// TIA Portal V16 program export: 1 tag tables, 12 data types, 26 data blocks, 18 code blocks (in call order from the OBs), 1 instance data blocks

VAR_GLOBAL   // PLC tag table "Default tag table"
   io_a AT %I0.0 : Bool;
   io_b AT %I0.1 : Bool;
END_VAR
VAR_GLOBAL CONSTANT   // user constants
   MAX_RPM : Int := 2800;
END_VAR

TYPE "SensorCommand"
VERSION : 0.1
   STRUCT
      enable { ExternalAccessible := 'False'; ExternalVisible := 'False'; ExternalWritable := 'False'} : Bool;
      mute { ExternalAccessible := 'False'; ExternalVisible := 'False'; ExternalWritable := 'False'} : Bool;
      case { ExternalAccessible := 'False'; ExternalVisible := 'False'; ExternalWritable := 'False'} : Int;
   END_STRUCT;

END_TYPE

TYPE "AnonStruct"
VERSION : 0.1
   STRUCT
      command : Struct
         a : Bool;
         b : Bool;
         c : Bool;
         others : Struct
            x : Bool;
            y : Bool;
            z : Bool := true;   // Definitely keep this one on.
         END_STRUCT;
      END_STRUCT;
   END_STRUCT;

END_TYPE

TYPE "ArrayWithDefault"
VERSION : 0.1
   STRUCT
      v : Array[0..15] of Bool := [false, true];
   END_STRUCT;

END_TYPE

TYPE "Pointf"
VERSION : 0.1
   STRUCT
      x : Real;
      y : Real;
   END_STRUCT;

END_TYPE

TYPE "Pointi"
VERSION : 0.1
   STRUCT
      x : Int;
      y : Int;
   END_STRUCT;

END_TYPE

TYPE "Polygon"
VERSION : 0.1
   STRUCT
      vertices { S7_SetPoint := 'False'} : Array[0..9] of "Pointi";   // Fixed size array
      n { S7_SetPoint := 'True'} : Int;   // of which this many points are valid
   END_STRUCT;

END_TYPE

TYPE "AppControl"
VERSION : 0.1
   STRUCT
      start : Bool;
      stop : Bool;
   END_STRUCT;

END_TYPE

TYPE "Box"
VERSION : 0.1
   STRUCT
      min { S7_SetPoint := 'False'} : "Point";
      max { S7_SetPoint := 'False'} : "Point";
   END_STRUCT;

END_TYPE

TYPE "MachineState"
VERSION : 0.1
   STRUCT
      running : Bool;
      faulted : Bool;
   END_STRUCT;

END_TYPE

TYPE "Point"
VERSION : 0.1
   STRUCT
      x : Int;
      y : Int;
   END_STRUCT;

END_TYPE

TYPE "SensorControl"
VERSION : 0.1
   STRUCT
      request_mode : Int;
   END_STRUCT;

END_TYPE

TYPE "SensorState"
VERSION : 0.1
   STRUCT
      mode : Int;
      ready : Bool;
   END_STRUCT;

END_TYPE

DATA_BLOCK "FromSafety"   // DB3
{ S7_Optimized_Access := 'TRUE' }
VERSION : 0.1
// stored: AutoNumber true, DBAccessibleFromOPCUA true, IsOnlyStoredInLoadMemory false, IsRetainMemResEnabled false, IsWriteProtectedInAS false, MemoryReserve 100
   VAR
      stop : Bool;
   END_VAR
BEGIN
END_DATA_BLOCK

DATA_BLOCK "ToSafety"   // DB2
{ S7_Optimized_Access := 'TRUE' }
VERSION : 0.1
// stored: AutoNumber true, DBAccessibleFromOPCUA true, IsOnlyStoredInLoadMemory false, IsRetainMemResEnabled false, IsWriteProtectedInAS false, MemoryReserve 100
   VAR
      "a" : Bool;
      "b" : Bool;
   END_VAR
BEGIN
END_DATA_BLOCK

DATA_BLOCK "DebugData"
{ S7_Optimized_Access := "TRUE" }
VERSION: 0.1
NON_RETAIN
    VAR
        source { ExternalAccessible := 'False'; ExternalVisible := 'False'; ExternalWritable := 'False'} : Int;
        flag : Bool;
    END_VAR

BEGIN
    source := 1;

END_DATA_BLOCK

DATA_BLOCK "AnonTestDB"
{ S7_Optimized_Access := 'TRUE' }
VERSION : 0.1
NON_RETAIN
   VAR 
      a { S7_SetPoint := 'False'} : "AnonStruct";
      b : "AnonStruct";   // custom comment for b
   END_VAR


BEGIN

END_DATA_BLOCK

DATA_BLOCK "PolygonDB"
{ S7_Optimized_Access := 'TRUE' }
VERSION : 0.1
NON_RETAIN
"Polygon"

BEGIN
   vertices[0].x := 0;
   vertices[0].y := 0;

END_DATA_BLOCK

DATA_BLOCK "DataFromSafety"
{ S7_Optimized_Access := 'TRUE' }
VERSION : 0.1
NON_RETAIN
   VAR 
      running : Bool;
   END_VAR


BEGIN

END_DATA_BLOCK

DATA_BLOCK "DataToSafety"
{ S7_Optimized_Access := 'TRUE' }
VERSION : 0.1
NON_RETAIN
   VAR 
      run : Bool;
   END_VAR


BEGIN

END_DATA_BLOCK

DATA_BLOCK "Main_Safety_RTG1_DB"
{ S7_Optimized_Access := 'TRUE' }
NAME : FUSI
VERSION : 0.1
NON_RETAIN
"Main_Safety_RTG1"

BEGIN

END_DATA_BLOCK

DATA_BLOCK "BlockIncrementer_DB"
{ S7_Optimized_Access := 'TRUE' }
VERSION : 0.1
NON_RETAIN
"BlockIncrementer"

BEGIN

END_DATA_BLOCK

DATA_BLOCK "MyCounter_DB0"
{ S7_Optimized_Access := 'TRUE' }
VERSION : 0.1
NON_RETAIN
"MyCounter"

BEGIN

END_DATA_BLOCK

DATA_BLOCK "MyCounter_DB1"
{ S7_Optimized_Access := 'TRUE' }
VERSION : 0.1
NON_RETAIN
"MyCounter"

BEGIN

END_DATA_BLOCK

DATA_BLOCK "Box"
{ S7_Optimized_Access := 'TRUE' }
VERSION : 0.1
NON_RETAIN
"Box"

BEGIN
   min.x := 0;

END_DATA_BLOCK

DATA_BLOCK "Example1_DB"
{ S7_Optimized_Access := 'TRUE' }
VERSION : 0.1
NON_RETAIN
   VAR 
      box0 { S7_SetPoint := 'False'} : "Box";
      box1 : "Box";
   END_VAR


BEGIN

END_DATA_BLOCK

DATA_BLOCK "Example2_DB"
{ S7_Optimized_Access := 'TRUE' }
VERSION : 0.1
NON_RETAIN
   VAR 
      reference { ExternalAccessible := 'False'; ExternalVisible := 'False'; ExternalWritable := 'False'; S7_SetPoint := 'False'} : "Point";
   END_VAR


BEGIN
   reference.x := 0;
   reference.y := 1;

END_DATA_BLOCK

DATA_BLOCK "F_SystemInfo_DB"
{ S7_Optimized_Access := 'TRUE' }
NAME : F_GLOBDB
VERSION : 0.1
NON_RETAIN
   VAR 
      FCCValue : DWord;
   END_VAR


BEGIN

END_DATA_BLOCK

DATA_BLOCK "RTG1SysInfo"
{InstructionName := 'F_CTRL1';
 LibVersion := '2.2';
 S7_Optimized_Access := 'TRUE' }
AUTHOR : SafeSys
FAMILY : F_CTRL
NAME : F_CTRL_1
VERSION : 2.2
NON_RETAIN
F_CTRL1

BEGIN
   F_SYSINFO.F_PROG_SIG := DW#16#832DEE38;
   F_SYSINFO.F_PROG_DAT := DTL#2021-8-4-22:50:56.862582800;
   F_SYSINFO.F_RTG_SIG := DW#16#F5BD20EF;
   F_SYSINFO.F_RTG_DAT := DTL#2021-8-4-22:50:56.862582800;
   F_SYSINFO.VERS_S7SAF := DW#16#16000000;
   dnMODE_C := 19127;
   dnDB_INIT_C := 70557;
   dnMOD_MODE_C := 34321;
   dnPLCSIM_MODE_C := 20664;
   dnACT_MOD_MODE_C := 27190;
   lnDIFF_C := 35673;
   lnDIFF_MTIME_C := 22975;
   nMAX_CYC := 120;
   dnMAX_CYC_C := 3819182;
   nWARN_CYC := 110;
   dwFCC_VALUE := DW#16#B0695B45;
   dnS_TIM_C := 14080;
   dnS_TIM_ALT_C := 33803;
   dnS_TIM100_CACHE_C := 32709;
   dnS_TIM100_USE_C := 25382;
   dnS_TIM1000_CACHE_C := 26562;
   dnS_TIM1000_USE_C := 41245;
   dnS_DIFF_C := 14080;
   dnS_DIFF100_C := 14080;
   dnS_DIFF1000_C := 14080;
   lnF_TIM_SFC_C := 14080;
   lnF_TIM_SFC_ALT_C := 27889;
   dnF_TIM_C := 14080;
   dnF_TIM_ALT_C := 23998;
   dnF_TIM100_CACHE_C := 26848;
   dnF_TIM100_USE_C := 25044;
   dnF_TIM1000_CACHE_C := 25507;
   dnF_TIM1000_USE_C := 23558;
   dnF_DIFF_C := 14080;
   dnF_DIFF100_C := 14080;
   dnF_DIFF1000_C := 14080;
   dnCONTROL_TIM100_C := 39214;
   dnCONTROL_TIM1000_C := 24463;
   dnTOL_C := 14080;
   dwF_PROG_SIG_DAT_SIG := DW#16#B04411D9;
   dwF_RTG_SIG_DAT_SIG := DW#16#C6D4DF0E;
   wRTG_NO := W#16#1;

END_DATA_BLOCK

DATA_BLOCK "DB1_C"
{ S7_Optimized_Access := 'TRUE' }
NAME : FCDI
VERSION : 0.1
NON_RETAIN
"FB1_C"

BEGIN
   dnCALLCHECK_C := 61159;
   dnTRACER_START := 20389;
   dnGCTX_DBNUMBER := 30010;

END_DATA_BLOCK

DATA_BLOCK "DB3_C"
{ S7_Optimized_Access := 'TRUE' }
NAME : FCDI
VERSION : 0.1
NON_RETAIN
"FB2_C"

BEGIN
   increment_C := 111444;
   counter_C := 92146;
   dnCALLCHECK_C := 87957;
   dnTRACER_START := 20944;
   dnGCTX_DBNUMBER := 30011;

END_DATA_BLOCK

DATA_BLOCK "DB4_C"
{ S7_Optimized_Access := 'TRUE' }
NAME : FCDI
VERSION : 0.1
NON_RETAIN
"FB2_C"

BEGIN
   increment_C := 138146;
   counter_C := 118848;
   dnCALLCHECK_C := 114659;
   dnTRACER_START := 20944;
   dnGCTX_DBNUMBER := 30011;

END_DATA_BLOCK

DATA_BLOCK "FB1_C_GCTX_DB"
{ S7_Optimized_Access := 'TRUE' }
NAME : F_GLOBDB
VERSION : 0.1
NON_RETAIN
   VAR 
      GCTX_DINT { ExternalAccessible := 'False'; ExternalVisible := 'False'; ExternalWritable := 'False'} : Array[0..0, 0..4] of DInt;
   END_VAR


BEGIN
   GCTX_DINT[0,0] := 1885684513;
   GCTX_DINT[0,1] := 32;
   GCTX_DINT[0,2] := 13215;
   GCTX_DINT[0,3] := 64;
   GCTX_DINT[0,4] := 96;

END_DATA_BLOCK

DATA_BLOCK "FB2_C_GCTX_DB"
{ S7_Optimized_Access := 'TRUE' }
NAME : F_GLOBDB
VERSION : 0.1
NON_RETAIN
   VAR 
      GCTX_DINT { ExternalAccessible := 'False'; ExternalVisible := 'False'; ExternalWritable := 'False'} : Array[0..2, 0..0] of DInt;
   END_VAR


BEGIN
   GCTX_DINT[0,0] := 1885664965;
   GCTX_DINT[1,0] := 19548;
   GCTX_DINT[2,0] := 1885684513;

END_DATA_BLOCK

DATA_BLOCK "FB32770_IDB_C"
{InstructionName := 'F_CTRLD';
 LibVersion := '1.4';
 S7_Optimized_Access := 'TRUE' }
AUTHOR : SafeSys
FAMILY : F_CTRL
NAME : F_CTRL_D
VERSION : 1.2
NON_RETAIN
F_CTRLD

BEGIN

END_DATA_BLOCK

DATA_BLOCK "FB32771_IDB_C"
{InstructionName := 'F_CTRL2';
 LibVersion := '1.4';
 S7_Optimized_Access := 'TRUE' }
AUTHOR : SafeSys
FAMILY : F_CTRL
NAME : F_CTRL_2
VERSION : 1.2
NON_RETAIN
F_CTRL2

BEGIN
   dnMOD_MODE_C := 55467;
   dnP_FOB := 8966;
   wRTG_NO := W#16#1;

END_DATA_BLOCK

DATA_BLOCK "FB32772_IDB_C"
{InstructionName := 'F_ETLI';
 LibVersion := '2.0';
 S7_Optimized_Access := 'TRUE' }
AUTHOR : SafeSys
FAMILY : F_CTRL
NAME : F_ET_LI
VERSION : 2.0
NON_RETAIN
F_ETLI

BEGIN

END_DATA_BLOCK

DATA_BLOCK "FB32773_IDB_C"
{InstructionName := 'F_CTRLRT';
 LibVersion := '1.3';
 S7_Optimized_Access := 'TRUE' }
AUTHOR : SafeSys
FAMILY : F_CTRL
NAME : F_CTRLRT
VERSION : 1.0
NON_RETAIN
F_CTRLRT

BEGIN

END_DATA_BLOCK

DATA_BLOCK "FOB_RTG1_GCTX_DB"
{ S7_Optimized_Access := 'TRUE' }
NAME : F_GLOBDB
VERSION : 0.1
NON_RETAIN
   VAR 
      GCTX_DINT { ExternalAccessible := 'False'; ExternalVisible := 'False'; ExternalWritable := 'False'} : Array[0..0, 0..2] of DInt;
   END_VAR


BEGIN
   GCTX_DINT[0,0] := 1885670433;
   GCTX_DINT[0,1] := 32;
   GCTX_DINT[0,2] := 8609;

END_DATA_BLOCK

ORGANIZATION_BLOCK "Main"   // OB1, LAD, ProgramCycle
TITLE = "Main Program Sweep (Cycle)"
{ S7_Optimized_Access := 'TRUE' }
VERSION : 0.1
// stored: AutoNumber true, IsIECCheckEnabled false, SetENOAutomatically false
   VAR_INPUT
      Initial_Call : Bool;   // Initial call of this OB
      Remanence : Bool;   // =True, if remanent data are available
   END_VAR
BEGIN
END_ORGANIZATION_BLOCK

FUNCTION_BLOCK "Main_Safety_RTG1"   // FB1, F_FBD
{ S7_Optimized_Access := 'TRUE' }
VERSION : 0.1
// stored: AutoNumber false, IsIECCheckEnabled false, UDAEnableTagReadback false
   VAR
      a_and_b : Bool;
      a_or_b : Bool;
      p_trig_state : Bool;
   END_VAR
   VAR_TEMP
      rising_a_or_b : Bool;
   END_VAR
   VAR_TEMP   // added for the SCL form of the ladder/FBD networks
      _w1 : Bool;
   END_VAR
BEGIN

REGION Network 1
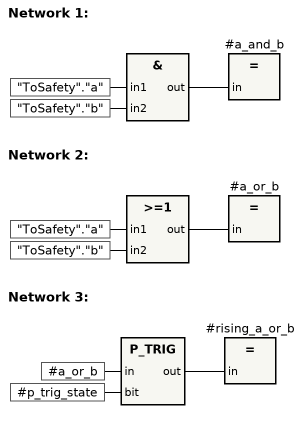
   #a_and_b := "ToSafety"."a" AND "ToSafety"."b";
END_REGION

REGION Network 2
   #a_or_b := "ToSafety"."a" OR "ToSafety"."b";
END_REGION

REGION Network 3
   #_w1 := #a_or_b AND NOT #p_trig_state;   // rising edge
   #p_trig_state := #a_or_b;
   #rising_a_or_b := #_w1;
END_REGION
END_FUNCTION_BLOCK

FUNCTION_BLOCK "Block_1"   // FB2, F_FBD
{ S7_Optimized_Access := 'TRUE' }
VERSION : 0.1
// stored: AutoNumber true, IsIECCheckEnabled false, UDAEnableTagReadback false
   VAR_INPUT
      "a" : Bool;
   END_VAR
   VAR_OUTPUT
      out0 : Bool;
      out1 : Bool;
   END_VAR
   VAR_TEMP
      t0 : Bool;
      ton : Bool;
   END_VAR
   VAR CONSTANT
      ALWAYS_FALSE : Bool := false;
   END_VAR
BEGIN

REGION Network 1
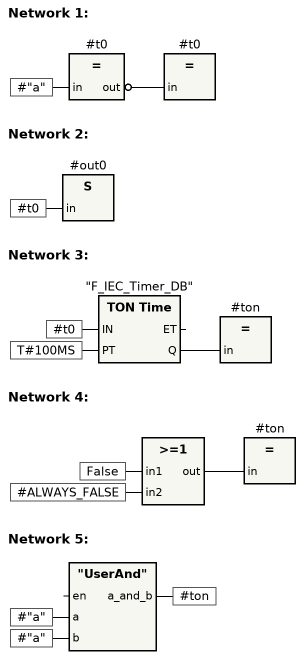
   #t0 := #"a";
   #t0 := NOT #"a";
END_REGION

REGION Network 2
   IF #t0 THEN #out0 := TRUE; END_IF;
END_REGION

REGION Network 3
   "F_IEC_Timer_DB".TON(IN := #t0, PT := T#100MS);
   #ton := "F_IEC_Timer_DB".Q;
END_REGION

REGION Network 4
   #ton := False OR #ALWAYS_FALSE;
END_REGION

REGION Network 5
   "UserAnd"("a" := #"a", "b" := #"a", a_and_b => #ton);
END_REGION
END_FUNCTION_BLOCK

FUNCTION "UserAnd" : Void   // FC1, F_FBD
{ S7_Optimized_Access := 'TRUE' }
VERSION : 0.1
// stored: AutoNumber true, IsIECCheckEnabled false, UDAEnableTagReadback false
   VAR_INPUT
      "a" : Bool;
      "b" : Bool;
   END_VAR
   VAR_OUTPUT
      a_and_b : Bool;
   END_VAR
BEGIN

REGION Network 1
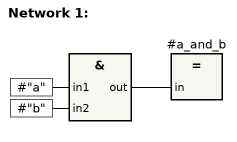
   #a_and_b := #"a" AND #"b";
END_REGION
END_FUNCTION

FUNCTION_BLOCK "DoubleAnd"   // FB3, F_FBD
{ S7_Optimized_Access := 'TRUE' }
VERSION : 0.1
// stored: AutoNumber true, IsIECCheckEnabled false, UDAEnableTagReadback false
   VAR_INPUT
      "a" : Bool;
      "b" : Bool;
      c : Bool;
      d : Bool;
   END_VAR
   VAR_OUTPUT
      i : Bool;
      j : Bool;
   END_VAR
BEGIN

REGION Network 1
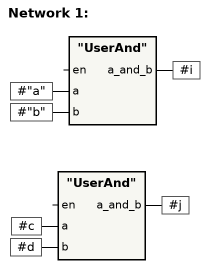
   "UserAnd"("a" := #"a", "b" := #"b", a_and_b => #i);
   "UserAnd"("a" := #c, "b" := #d, a_and_b => #j);
END_REGION
END_FUNCTION_BLOCK

FUNCTION "UserSet" : Void   // FC3, F_FBD
{ S7_Optimized_Access := 'TRUE' }
VERSION : 0.1
// stored: AutoNumber true, IsIECCheckEnabled false, UDAEnableTagReadback false
   VAR_INPUT
      q : Bool;
   END_VAR
   VAR_IN_OUT
      "a" : Bool;
   END_VAR
BEGIN

REGION Network 1
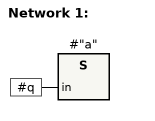
   IF #q THEN #"a" := TRUE; END_IF;
END_REGION
END_FUNCTION

FUNCTION "NoOp" : Void   // FC4, F_FBD
{ S7_Optimized_Access := 'TRUE' }
VERSION : 0.1
// stored: AutoNumber true, IsIECCheckEnabled false, UDAEnableTagReadback false
   VAR_IN_OUT
      "a" : Bool;
   END_VAR
BEGIN
END_FUNCTION

FUNCTION "TestSuite" : Void   // FC6, F_FBD
{ S7_Optimized_Access := 'TRUE' }
VERSION : 0.1
// stored: AutoNumber true, IsIECCheckEnabled false, UDAEnableTagReadback false
   VAR_IN_OUT
      test_nop_var : Bool;
   END_VAR
BEGIN

REGION Network 1: Test No-Op
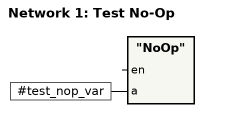
   "NoOp"("a" := #test_nop_var);
END_REGION
END_FUNCTION

FUNCTION_BLOCK "UserAdd"   // FB4, F_FBD
{ S7_Optimized_Access := 'TRUE' }
VERSION : 0.1
// stored: AutoNumber true, IsIECCheckEnabled false, UDAEnableTagReadback false
   VAR_TEMP
      "a" : Int;
      "b" : Int;
      result : Int;
   END_VAR
BEGIN

REGION Network 1
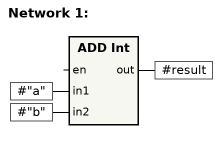
   #result := #"a" + #"b";
END_REGION
END_FUNCTION_BLOCK

FUNCTION "UserSetTest" : Void   // FC5, F_FBD
{ S7_Optimized_Access := 'TRUE' }
VERSION : 0.1
// stored: AutoNumber true, IsIECCheckEnabled false, UDAEnableTagReadback false
   VAR_TEMP
      "a" : Bool;
      q : Bool;
   END_VAR
BEGIN

REGION Network 1
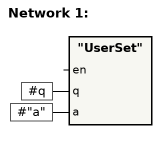
   "UserSet"(q := #q, "a" := #"a");
END_REGION
END_FUNCTION

FUNCTION "Demo" : Void   // FC2, F_FBD
{ S7_Optimized_Access := 'TRUE' }
VERSION : 0.1
// stored: AutoNumber true, IsIECCheckEnabled false, UDAEnableTagReadback false
   VAR_INPUT
      is_slow : Bool;
      left_clear : Bool;
      right_clear : Bool;
      mute_req : Bool;
      estop_clear : Bool;
   END_VAR
   VAR_OUTPUT
      stop : Bool;
   END_VAR
   VAR_TEMP
      mute_granted : Bool;
      scanners_ok : Bool;
   END_VAR
BEGIN

REGION Network 1
   // A mute request may be granted if the machine is moving slow enough to make it avoidable.
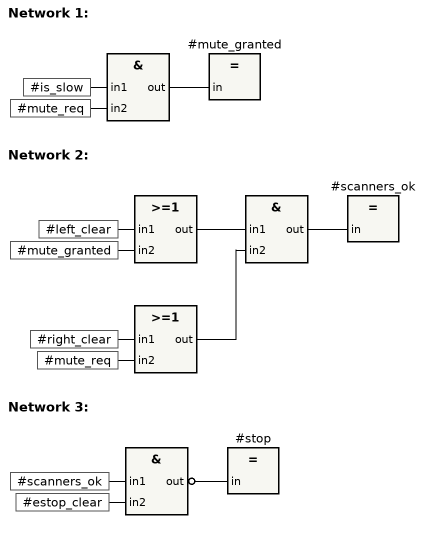
   #mute_granted := #is_slow AND #mute_req;
END_REGION

REGION Network 2
   // The safety scanner system evalutes the state of each safety field and condenses it to a single, overall status for the safety fields.
   #scanners_ok := (#left_clear OR #mute_granted) AND (#right_clear OR #mute_req);
END_REGION

REGION Network 3
   // Combine safety subsystems into a single stop variable
   #stop := NOT (#scanners_ok AND #estop_clear);
END_REGION
END_FUNCTION

FUNCTION "RunSensors" : Void   // FC8, F_FBD
{ S7_Optimized_Access := 'TRUE' }
VERSION : 0.1
// stored: AutoNumber true, IsIECCheckEnabled false, UDAEnableTagReadback false
   VAR_INPUT
      command_a : "SensorCommand";
      command_b : "SensorCommand";
   END_VAR
   VAR_OUTPUT
      all_ok : Bool;
      last_command_a : "SensorCommand";
   END_VAR
   VAR_TEMP
      a_ok : Bool;
      b_ok : Bool;
   END_VAR
BEGIN

REGION Network 1
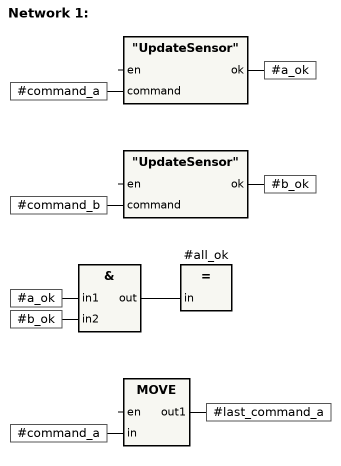
   "UpdateSensor"(command := #command_a, ok => #a_ok);
   "UpdateSensor"(command := #command_b, ok => #b_ok);
   #all_ok := #a_ok AND #b_ok;
   #last_command_a := #command_a;
END_REGION
END_FUNCTION

FUNCTION "UpdateSensor" : Void   // FC7, F_FBD
{ S7_Optimized_Access := 'TRUE' }
VERSION : 0.1
// stored: AutoNumber true, IsIECCheckEnabled false, UDAEnableTagReadback false
   VAR_INPUT
      command : "SensorCommand";
   END_VAR
   VAR_OUTPUT
      ok : Bool;
   END_VAR
BEGIN

REGION Network 1
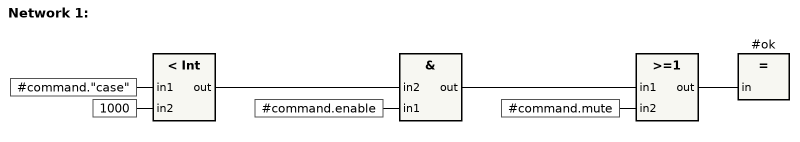
   #ok := ((#command."case" < 1000) AND #command.enable) OR #command.mute;
END_REGION
END_FUNCTION

FUNCTION_BLOCK "Step1"   // FB3, F_FBD
{ S7_Optimized_Access := 'TRUE' }
VERSION : 0.1
// stored: AutoNumber true, IsIECCheckEnabled false, UDAEnableTagReadback false
BEGIN

REGION Network 1
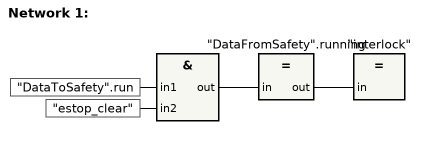
   "DataFromSafety".running := "DataToSafety".run AND "estop_clear";
   "interlock" := "DataFromSafety".running;
END_REGION
END_FUNCTION_BLOCK

FUNCTION_BLOCK "Step2"   // FB2, F_FBD
{ S7_Optimized_Access := 'TRUE' }
VERSION : 0.1
// stored: AutoNumber true, IsIECCheckEnabled false, UDAEnableTagReadback false
   VAR
      faults_clear : Bool;
      last_estop_clear : Bool;
      last_reset : Bool;
   END_VAR
   VAR_TEMP   // added for the SCL form of the ladder/FBD networks
      _w1 : Bool;
      _w2 : Bool;
   END_VAR
BEGIN

REGION Network 1
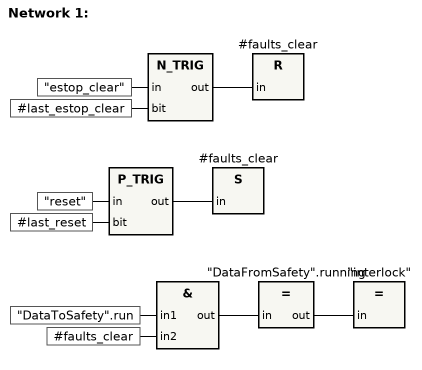
   #_w1 := NOT "estop_clear" AND #last_estop_clear;   // falling edge
   #last_estop_clear := "estop_clear";
   IF #_w1 THEN #faults_clear := FALSE; END_IF;
   #_w2 := "reset" AND NOT #last_reset;   // rising edge
   #last_reset := "reset";
   IF #_w2 THEN #faults_clear := TRUE; END_IF;
   "DataFromSafety".running := "DataToSafety".run AND #faults_clear;
   "interlock" := "DataFromSafety".running;
END_REGION
END_FUNCTION_BLOCK

FUNCTION_BLOCK "BlockIncrementer"   // FB3, F_FBD
{ S7_Optimized_Access := 'TRUE' }
VERSION : 0.1
// stored: AutoNumber true, IsIECCheckEnabled false, UDAEnableTagReadback false
   VAR
      "a" : "MyCounter";
      "b" : "MyCounter";
   END_VAR
BEGIN

REGION Network 1
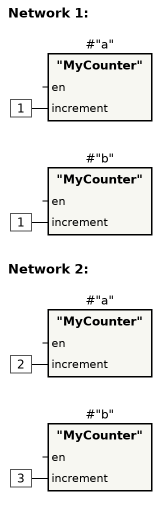
   #"a"(increment := 1);   // "MyCounter"
   #"b"(increment := 1);   // "MyCounter"
END_REGION

REGION Network 2
   #"a"(increment := 2);   // "MyCounter"
   #"b"(increment := 3);   // "MyCounter"
END_REGION
END_FUNCTION_BLOCK

FUNCTION_BLOCK "MyCounter"   // FB2, F_FBD
{ S7_Optimized_Access := 'TRUE' }
VERSION : 0.1
// stored: AutoNumber true, IsIECCheckEnabled false, UDAEnableTagReadback false
   VAR_INPUT
      increment : Int;
   END_VAR
   VAR
      "counter" : Int;
   END_VAR
BEGIN

REGION Network 1
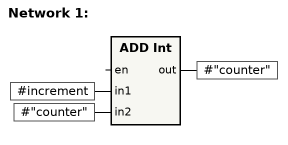
   #"counter" := #increment + #"counter";
END_REGION
END_FUNCTION_BLOCK

FUNCTION "ProcessSensor" : Void   // FC1, F_FBD
{ S7_Optimized_Access := 'TRUE' }
VERSION : 0.1
// stored: AutoNumber true, IsIECCheckEnabled false, UDAEnableTagReadback false
   VAR_INPUT
      ctrl : "SensorControl";
   END_VAR
   VAR_OUTPUT
      state : "SensorState";
      safe : Bool;
   END_VAR
BEGIN

REGION Network 1
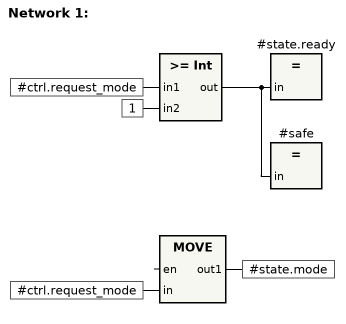
   #state.ready := #ctrl.request_mode >= 1;
   #safe := #state.ready;
   #state.mode := #ctrl.request_mode;
END_REGION
END_FUNCTION

DATA_BLOCK "Main_Safety_RTG1_DB"   // DB1, F_DB
NAME : FUSI
VERSION : 0.1
// stored: AutoNumber true, DBAccessibleFromOPCUA true, InstanceOfName Main_Safety_RTG1, InstanceOfType FB
"Main_Safety_RTG1"
BEGIN
END_DATA_BLOCK
